Staubli VAL3: gestureWaveIn.pgx

program gestureWaveIn()
begin
  putln("WaveInCAlled")
  joint1TestCopy = joint1Test
  movej(joint1Test,tClaw,nom_speed)
end
